(* IEC 61131-3 sources: programs/VI-54/VI-54_20171205/VI-54_20171205/Stations/Screen/LseClass170718/Class/GiveConfigNumber, 1 file *)

(* ---- GiveConfigNumber.st ---- *)
(*!
<Class
	Name               = "GiveConfigNumber"
	Revision           = "1.0"
	RealtimeTask       = "false"
	CyclicTask         = "false"
	BackgroundTask     = "false"
	Sigmatek           = "false"
	OSInterface        = "false"
	HighPriority       = "false"
	Automatic          = "false"
	UpdateMode         = "Prescan"
	SharedCommandTable = "true"
	Objectsize         = "(376,120)">
	<Channels>
		<Server Name="GroupNbr" Visualized="false" Initialize="false" WriteProtected="true" Retentive="false"/>
		<Server Name="Next" Visualized="false" Initialize="false" WriteProtected="false" Retentive="false"/>
		<Server Name="Nmb1" Visualized="false" Initialize="false" WriteProtected="true" Retentive="false"/>
		<Server Name="Nmb10" Visualized="false" Initialize="false" WriteProtected="true" Retentive="false"/>
		<Server Name="Nmb11" Visualized="false" Initialize="false" WriteProtected="true" Retentive="false"/>
		<Server Name="Nmb12" Visualized="false" Initialize="false" WriteProtected="true" Retentive="false"/>
		<Server Name="Nmb13" Visualized="false" Initialize="false" WriteProtected="true" Retentive="false"/>
		<Server Name="Nmb14" Visualized="false" Initialize="false" WriteProtected="true" Retentive="false"/>
		<Server Name="Nmb15" Visualized="false" Initialize="false" WriteProtected="true" Retentive="false"/>
		<Server Name="Nmb16" Visualized="false" Initialize="false" WriteProtected="true" Retentive="false"/>
		<Server Name="Nmb2" Visualized="false" Initialize="false" WriteProtected="true" Retentive="false"/>
		<Server Name="Nmb3" Visualized="false" Initialize="false" WriteProtected="true" Retentive="false"/>
		<Server Name="Nmb4" Visualized="false" Initialize="false" WriteProtected="true" Retentive="false"/>
		<Server Name="Nmb5" Visualized="false" Initialize="false" WriteProtected="true" Retentive="false"/>
		<Server Name="Nmb6" Visualized="false" Initialize="false" WriteProtected="true" Retentive="false"/>
		<Server Name="Nmb7" Visualized="false" Initialize="false" WriteProtected="true" Retentive="false"/>
		<Server Name="Nmb8" Visualized="false" Initialize="false" WriteProtected="true" Retentive="false"/>
		<Server Name="Nmb9" Visualized="false" Initialize="false" WriteProtected="true" Retentive="false"/>
		<Client Name="Group" Required="false" Internal="false"/>
		<Client Name="Number" Required="false" Internal="false"/>
	</Channels>
</Class>
*)
GiveConfigNumber : CLASS
  //Servers:
	Nmb1 	: SvrChCmd_DINT;
	Nmb2 	: SvrCh_DINT;
	Nmb3 	: SvrCh_DINT;
	Nmb4 	: SvrCh_DINT;
	Nmb5 	: SvrCh_DINT;
	Nmb6 	: SvrCh_DINT;
	Nmb7 	: SvrCh_DINT;
	Nmb8 	: SvrCh_DINT;
	Nmb9 	: SvrCh_DINT;
	Nmb10 	: SvrCh_DINT;
	Nmb11 	: SvrCh_DINT;
	Nmb12 	: SvrCh_DINT;
	Nmb13 	: SvrCh_DINT;
	Nmb14 	: SvrCh_DINT;
	Nmb15 	: SvrCh_DINT;
	Nmb16 	: SvrCh_DINT;
	GroupNbr 	: SvrCh_DINT;
	Next 	: SvrCh_DINT;
  //Clients:
	Number 	: CltChCmd__16Alarms;
	Group 	: CltCh_DINT;
  //Variables:
  //Functions:

	FUNCTION VIRTUAL GLOBAL Init;
  //Tables:
	FUNCTION @STD
		VAR_OUTPUT
			ret_code	: CONFSTATES;
		END_VAR;
	FUNCTION GLOBAL TAB @CT_;
END_CLASS;

#pragma usingLtd _16Alarms

FUNCTION VIRTUAL GLOBAL GiveConfigNumber::Init

  Number := Next.Read();
  If Number < 0 then
    Number := 0;
  end_if;

  Nmb1 := Number;
  Nmb2 := Nmb1 + 1;
  Nmb3 := Nmb2 + 1;
  Nmb4 := Nmb3 + 1;
  Nmb5 := Nmb4 + 1;
  Nmb6 := Nmb5 + 1;
  Nmb7 := Nmb6 + 1;
  Nmb8 := Nmb7 + 1;
  Nmb9 := Nmb8 + 1;
  Nmb10 := Nmb9 + 1;
  Nmb11 := Nmb10 + 1;
  Nmb12 := Nmb11 + 1;
  Nmb13 := Nmb12 + 1;
  Nmb14 := Nmb13 + 1;
  Nmb15 := Nmb14 + 1;
  Nmb16 := Nmb15 + 1;

  //Next  := Nmb16 + 1;
  if IsClientConnected(#Number) then
    Number.Next.Write(input:= Nmb16 + 1);
  end_if;

  Group := Group.Read();
  GroupNbr := Group;

END_FUNCTION
